{attribute 'GeneratedUsingTerminal: EP5001-0002-0016'}
{attribute addProperty BoxType "EP5001-0002-0016"}
{attribute addProperty Id "StatusAT %I*Status_ACC8459F6Counter_valueAT %I*UDINT4"}
{attribute addProperty CRC "238915123"}
{attribute addProperty Size "10"}
TYPE SSI_Inputs_0E3D8E33 EXTENDS InputBase_8311D824 :
STRUCT
	{attribute addProperty Name "Status"}
	Status AT %I* : Status_ACC8459F;
	{attribute addProperty Name "Counter_value"}
	Counter_value AT %I* : UDINT;
END_STRUCT
END_TYPE

(* stored: Version 1.2.0.0, ProductVersion 3.1.4024.11
   DUT SSI_Inputs_0E3D8E33: Id {e4892f38-b347-41b5-9805-0b3456241a3b} *)
